TYPE
	NW_BUF_SHORT : ARRAY[0..NETWORK_BUFFER_SHORT_SIZE] OF BYTE;
END_TYPE

(* stored: Version 1.1.0.1, ProductVersion 3.1.4024.4
   DUT NW_BUF_SHORT: Id {00ebc2ff-04b6-4e0a-96ba-2d6baf76517f} *)
